// TIA Portal V19 export
DATA_BLOCK "PPrgArchive12"   // DB511
// stored: IsOnlyStoredInLoadMemory true, MemoryReserve 0, Namespace G
   VAR RETAIN
      PRG : Array[1101..1200] of "PPrg_Data";
   END_VAR
BEGIN
END_DATA_BLOCK
